(* IEC 61131-3 sources: repolevel_ST_code_completion/output/0122完整版本_无planner目前sota/repoeval_counter/readful_result_no_provide, 1 file *)

(* ---- FB_counter.st ---- *)
VAR
    nPrevValue: INT;    (*存储之前的数值*)
END_VAR

IF bReset THEN
    nValue := 0;        (*数据清零*)
ELSIF bUp THEN
    nValue := nValue + 1; (*数据递增*)
ELSIF bDown THEN
    nValue := nValue - 1; (*数据递减*)
END_IF

nPrevValue := nValue;    (*更新之前的数值*)
END_FUNCTION_BLOCK
